RESOURCE_TYPE TESTPAR_RES (* Test Java generation of FB parameters in a resource type. *)
  (* Standard: 61499-1 *)
  (* Version 0.0, 2004-12-16, JHC, Rockwell Automation *)
  (* Compiler header: package fb.rt.test; import fb.rt.math.*; import fb.rt.net.*; *)
  (* Compiler Java Sun JDK 1.4.2 *)
  VAR_INPUT
    SUBSC_ID : WSTRING;
    PUBL_ID : WSTRING;
  END_VAR
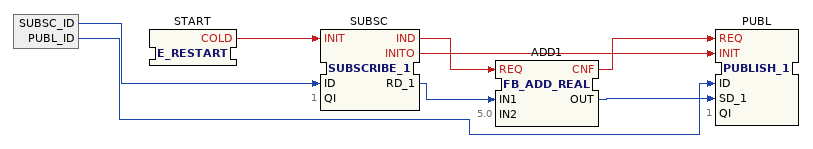
  FBS
    START : E_RESTART;
    ADD1 : FB_ADD_REAL(IN2 := 5.0);
    SUBSC : SUBSCRIBE_1(QI := 1);
    PUBL : PUBLISH_1(QI := 1);
  END_FBS
  EVENT_CONNECTIONS
    START.COLD TO SUBSC.INIT;
    SUBSC.IND TO ADD1.REQ;
    ADD1.CNF TO PUBL.REQ;
    SUBSC.INITO TO PUBL.INIT;
  END_CONNECTIONS
  DATA_CONNECTIONS
    SUBSC_ID TO SUBSC.ID;
    SUBSC.RD_1 TO ADD1.IN1;
    PUBL_ID TO PUBL.ID;
    ADD1.OUT TO PUBL.SD_1;
  END_CONNECTIONS
END_RESOURCE_TYPE
